Staubli VAL3: onStart.pgx

program onStart()
  local num i
  local string l_sMessage
begin
  // reset the index
  nIndex=nSelected=nView=0
  // reset the Key pressure
  call use:nullKey(nKey)
  // logMsg
  logMsg("[KERNEL] INTERFACE:PAGE view program")
  //
  sProgram=sItems[0]
  //
  call prog:load(sProgram,i)
  if i!=0
// error loading
    call language:message(l_sMessage,-7)
    popUpMsg(l_sMessage+" PROG "+sProgram+" code "+toString("",i))
  endIf
  // define the list
  call buildList()
  // build the page
  call refreshStatic()
  logMsg("ON MEMORY events INSTRUCTION "+events:libPath())
end
